// TIA Portal V19 export
TYPE "LEXCHANGETRAY_typeRoller_toWorkstationDeliver_B2"
// stored: Access Published
   STRUCT
      feedback : "LEXCHANGETRAY_typeRoller_toWorkStationRollerFeedback_B2";
      req { S7_SetPoint := 'True'} : "LEXCHANGETRAY_typeRoller_toWorkStationRollerReq_B2";
   END_STRUCT;
END_TYPE
